# EPICS substitutions: vacuum/MAIN_TRUNK/vacApp/Db/l407_agilent4uhv.substitutions
# Agilent4UHV substitutions file

file db/agilent4uhv.db
{
     pattern {LOCA,			DEV,			PORT,		ADDR,	TIMEOUT}
     		{HL4,			VL407_1,		4uhv_1,		0,		0.2}
     		{HL4,			VL407_2,		4uhv_2,		0,		0.2}
}

file db/agilent4uhv_alias.db
{
     pattern {LOCA,			DEV,			SUB1,				SUB2,				SUB3,					SUB4,				PORT,		ADDR,	TIMEOUT}
     		 {HL4,			VL407_1,		IP01:L407_Acc601,		IP02:L407_Acc602,		IP03:L407_Acc603,			IP04:L407_Acc604,		4uhv_1,		0,		0.2}
		 {HL4,			VL407_2,		IP05:L407_Acc605,		IP06:L407_Wave601,	IP07:L407_Kly601,			IP08:Empty,			4uhv_2,		0,		0.2}
}
